// TIA Portal V20 export
DATA_BLOCK "ReceiveFData_BA30AC1"   // DB57
// stored: InstanceOfName Safety.GM_ReceiveFData, InstanceOfType FB, Namespace Safety
"Safety.GM_ReceiveFData"
   // VAR_INPUT
   //    Connection_ID_Send : Word;
   //    Connection_ID_Receive : Word;
   //    Send_Ack_Rcv_Length : UInt;
   //    Receive_Rcv_Length : UInt;
   // END_VAR
   // VAR_IN_OUT
   //    RcvBuffer : Array[0..1, 0..121] of Byte;
   //    ReceivedData : Array[0..121] of Byte;
   //    ReceivedAck : Array[0..121] of Byte;
   // END_VAR
   // VAR
   //    instTRcvAck { S7_SetPoint := 'True'} : TRCV;
   //    instTRcvData { S7_SetPoint := 'True'} : TRCV;
   //    statErrorRcvAck { S7_SetPoint := 'True'} : Word;
   //    statErrorRcvData : Word;
   // END_VAR
BEGIN
END_DATA_BLOCK
